(* CoDeSys 2.3 export: ADS_COMMUNICATION.EXP *)

(* POU ADS_Communication, CFC *)
PROGRAM ADS_Communication
VAR
	fb_DerevoADSwrite: ADSWRITE;
	fb_floor1ADSwrite: ADSWRITE;

	counter_error,counter_busy: CTU;
END_VAR
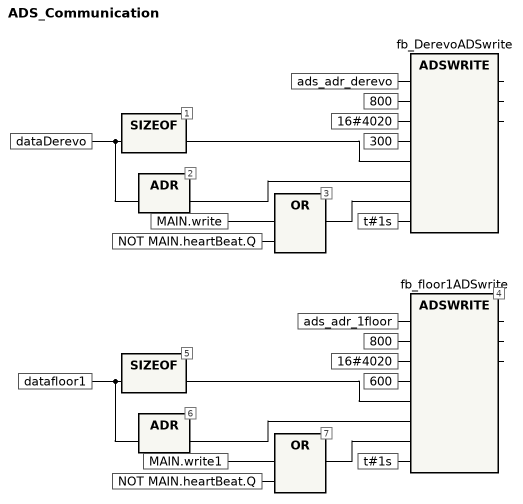
_CFC_ (* Continuous Function Chart, elements in execution order *)
#0 fb_DerevoADSwrite:ADSWRITE(ads_adr_derevo, 800, 16#4020, 300, #1, #2, #3, t#1s)
#1 SIZEOF(dataDerevo)
#2 ADR(dataDerevo)
#3 OR(MAIN.write, NOT MAIN.heartBeat.Q)
#4 fb_floor1ADSwrite:ADSWRITE(ads_adr_1floor, 800, 16#4020, 600, #5, #6, #7, t#1s)
#5 SIZEOF(datafloor1)
#6 ADR(datafloor1)
#7 OR(MAIN.write1, NOT MAIN.heartBeat.Q)
_END_CFC_
END_PROGRAM
